{attribute 'GeneratedUsingTerminal: EK1100-0000-0018'}
{attribute addProperty BoxType "EK1100-0000-0018"}
{attribute addProperty Id "Beckhoff_EP5xxxEK1122Beckhoff_EP5xxxEK1122_1DAC1461409"}
{attribute addProperty CRC "1809636415"}
{attribute addProperty Size "409"}
TYPE Beckhoff_EP5xxx_6BDCDC3F EXTENDS EK1100_AB5A9467 :
STRUCT
	{attribute addProperty Name "Beckhoff_EP5xxxEK1122"}
	Beckhoff_EP5xxxEK1122 : Beckhoff_EP5xxxEK1122_1DAC1461;
END_STRUCT
END_TYPE

(* stored: Version 1.2.0.0, ProductVersion 3.1.4024.9
   DUT Beckhoff_EP5xxx_6BDCDC3F: Id {5e43ee15-b317-42b5-9436-90ff7a8dff60} *)
